INTERFACE IPushoverClient

/// \copydoc Pushover.PushoverClient#Clear
METHOD Clear : IPushoverClient
END_METHOD

/// \copydoc Pushover.PushoverClient#EnableHtml
METHOD EnableHtml : IPushoverClient
END_METHOD

/// \copydoc Pushover.PushoverClient#EnableMonospace
METHOD EnableMonospace : IPushoverClient
END_METHOD

/// \copydoc Pushover.PushoverClient#SendMessageAsync
METHOD SendMessageAsync
VAR_IN_OUT CONSTANT
  title : STRING(255);
  message : STRING(255);
END_VAR
END_METHOD

/// \copydoc Pushover.PushoverClient#WithCallback
METHOD WithCallback : IPushoverClient
VAR_IN_OUT CONSTANT
  callback : STRING(255);
END_VAR
END_METHOD

/// \copydoc Pushover.PushoverClient#WithDevice
METHOD WithDevice : IPushoverClient
VAR_IN_OUT CONSTANT
  device : STRING(80);
END_VAR
END_METHOD

/// \copydoc Pushover.PushoverClient#WithExpire
METHOD WithExpire : IPushoverClient
VAR_INPUT
  expire : INT;
END_VAR
END_METHOD

/// \copydoc Pushover.PushoverClient#WithPriority
METHOD WithPriority : IPushoverClient
VAR_INPUT
  priority : PushoverPriority;
END_VAR
END_METHOD

/// \copydoc Pushover.PushoverClient#WithProxy
METHOD WithProxy : IPushoverClient
VAR_IN_OUT CONSTANT
  host : STRING(80);
END_VAR
VAR_INPUT
  port : INT;
END_VAR
END_METHOD

/// \copydoc Pushover.PushoverClient#WithRetry
METHOD WithRetry : IPushoverClient
VAR_INPUT
  retry : INT;
END_VAR
END_METHOD

/// \copydoc Pushover.PushoverClient#WithSound
METHOD WithSound : IPushoverClient
VAR_INPUT
  sound : PushoverSound;
END_VAR
END_METHOD

/// \copydoc Pushover.PushoverClient#WithTimestamp
METHOD WithTimestamp : IPushoverClient
VAR_INPUT
  timestamp : INT; //< UNIX Timestamp in seconds
END_VAR
END_METHOD

/// \copydoc Pushover.PushoverClient#WithTimeToLive
METHOD WithTimeToLive : IPushoverClient
VAR_INPUT
  ttl : INT; //< Seconds until this message should be automatically removed from the device. Needs to be positive
END_VAR
END_METHOD

/// \copydoc Pushover.PushoverClient#WithUrl
METHOD WithUrl : IPushoverClient
VAR_IN_OUT CONSTANT
  url : STRING(255);
END_VAR
END_METHOD

/// \copydoc Pushover.PushoverClient#WithUrlTitle
METHOD WithUrlTitle : IPushoverClient
VAR_IN_OUT CONSTANT
  urlTitle : STRING(255);
END_VAR
END_METHOD

END_INTERFACE

(* stored: Version 1.1.0.1, ProductVersion 3.1.4024.12
   Itf IPushoverClient: Id {1de1b2e7-821a-4c35-9e95-45170d4d91e5}
   Method Clear: Id {f8d769bc-0485-4d12-99e8-0093ee232421}
   Method EnableHtml: Id {6327050e-f9e5-4b5b-be12-d03a4472a486}
   Method EnableMonospace: Id {7a3a5331-2be1-41ce-a243-6efb60dac001}
   Method SendMessageAsync: Id {a43c981d-98f5-48cd-9610-5e013c2971cd}
   Method WithCallback: Id {a705da4b-d7a2-4587-b5b0-03876650e79b}
   Method WithDevice: Id {1e39f546-bb31-42d1-9cf0-e78e58fdc581}
   Method WithExpire: Id {eeef378d-2d3a-4f09-8994-9a2adb58a88b}
   Method WithPriority: Id {16481bc8-fc63-4c1c-a4c1-b6a435cd92ba}
   Method WithProxy: Id {0005b2dd-2a91-4f2b-b1d2-de942a828ef1}
   Method WithRetry: Id {3e25cabc-2ea7-42af-930a-9a1e1d333a75}
   Method WithSound: Id {1a16239a-44fd-4959-9987-4d9cbcdb3745}
   Method WithTimestamp: Id {d84a36b1-b9cb-4a1c-8e4d-615fb900f724}
   Method WithTimeToLive: Id {45053ff4-00b9-4cab-b692-cc7bba5d6db9}
   Method WithUrl: Id {ad9da46b-6f11-4121-8941-349cd26bfe70}
   Method WithUrlTitle: Id {cb56259a-2b95-4a0e-b09a-7bd29193e1b2} *)
